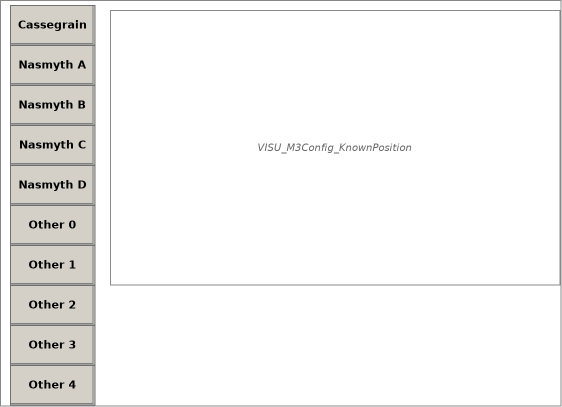
VISUALIZATION VISU_M3Config_KnownPositions  // 562x407
VAR_IN_OUT
	currentPosition : INT;
    active : M3KnownPositionsConfig;
    editable : M3KnownPositionsConfig;
END_VAR
    Frame (110,10 450x275), frame switch variable: currentPosition
        shows VISU_M3Config_KnownPosition(active := active.cassegrain, editable := editable.cassegrain)
        shows VISU_M3Config_KnownPosition(active := active.nasmythA, editable := editable.nasmythA)
        shows VISU_M3Config_KnownPosition(active := active.nasmythB, editable := editable.nasmythB)
        shows VISU_M3Config_KnownPosition(active := active.nasmythC, editable := editable.nasmythC)
        shows VISU_M3Config_KnownPosition(active := active.nasmythD, editable := editable.nasmythD)
        shows VISU_M3Config_KnownPosition(active := active.other0, editable := editable.other0)
        shows VISU_M3Config_KnownPosition(active := active.other1, editable := editable.other1)
        shows VISU_M3Config_KnownPosition(active := active.other2, editable := editable.other2)
        shows VISU_M3Config_KnownPosition(active := active.other3, editable := editable.other3)
        shows VISU_M3Config_KnownPosition(active := active.other4, editable := editable.other4)
        shows VISU_M3Config_KnownPosition(active := active.position9)
    Button (10,5 85x40), "Cassegrain", pressed state: currentPosition = 0
        OnMouseClick: execute { currentPosition := 0; }
    Button (10,45 85x40), "Nasmyth A", pressed state: currentPosition = 1
        OnMouseClick: execute { currentPosition := 1; }
    Button (10,85 85x40), "Nasmyth B", pressed state: currentPosition = 2
        OnMouseClick: execute { currentPosition := 2; }
    Button (10,125 85x40), "Nasmyth C", pressed state: currentPosition = 3
        OnMouseClick: execute { currentPosition := 3; }
    Button (10,165 85x40), "Nasmyth D", pressed state: currentPosition = 4
        OnMouseClick: execute { currentPosition := 4; }
    Button (10,205 85x40), "Other 0", pressed state: currentPosition = 5
        OnMouseClick: execute { currentPosition := 5; }
    Button (10,245 85x40), "Other 1", pressed state: currentPosition = 6
        OnMouseClick: execute { currentPosition := 6; }
    Button (10,285 85x40), "Other 2", pressed state: currentPosition = 7
        OnMouseClick: execute { currentPosition := 7; }
    Button (10,325 85x40), "Other 3", pressed state: currentPosition = 8
        OnMouseClick: execute { currentPosition := 8; }
    Button (10,365 85x40), "Other 4", pressed state: currentPosition = 9
        OnMouseClick: execute { currentPosition := 9; }
END_VISUALIZATION

(* stored: Version 1.1.0.1, ProductVersion 3.1.4019.2
   Visu VISU_M3Config_KnownPositions: Id {6db81f55-dab9-4ea3-ad5b-ab953eb1fae1} *)
